TYPE EL3356_RMB_Value :
STRUCT
	{attribute addProperty Name "Value"}
	Value AT %I* : DINT;
END_STRUCT
END_TYPE

(* stored: Version 1.1.0.1, ProductVersion 3.1.4024.9
   DUT EL3356_RMB_Value: Id {4aee517e-c70a-0314-2cf5-98775fb5b61a} *)
